PROGRAM io_mapping
VAR PERSISTENT
    //Example analog input function block
    cpt_3144 : analog_scaling;
	
	test_real AT %Q* : REAL;
	
	publisharray AT %Q* : ARRAY[0..9] OF REAL;
	
	sine_wave : REAL;
	
    //Example Analog input raw input, mapped to a physical input
    cpt_3144_raw_input AT %I* : INT;

END_VAR

//Instantiate Example analog input function block
cpt_3144();

//Map values from the OPC GVL so that they can be written to from outside POU(IE from HMI)
cpt_3144.eu_max:=opc.popa_0081_cpt_3144_eu_max;
cpt_3144.eu_min:=opc.popa_0081_cpt_3144_eu_min;
cpt_3144.filter_factor:=opc.popa_0081_cpt_3144_filter_factor;
cpt_3144.raw_max:=opc.popa_0081_cpt_3144_raw_max;
cpt_3144.raw_min:=opc.popa_0081_cpt_3144_raw_min;
//Map the analog scaling function block raw input to the physical raw input variable
cpt_3144.raw_input := cpt_3144_raw_input;

sine_wave:=sine_wave+0.001;
IF (sine_wave>(2*pi)) THEN
	sine_wave:=0;
END_IF

publisharray[0]:=sine_wave;
publisharray[1]:=sine_wave/2;
publisharray[2]:=sine_wave*2;

END_PROGRAM

(* stored: Version 1.1.0.1, ProductVersion 3.1.4024.12
   POU io_mapping: Id {87c33c1f-405d-4536-940a-0d0026912d98}, SpecialFunc None *)
